// This function has been automatically generated from the project information.
{attribute 'signature_flag' := '1073741824'}
{attribute 'TcGenerated'}
{attribute 'no-analysis'}
FUNCTION F_GetTitle : WSTRING
VAR_INPUT
	
END_VAR

F_GetTitle := "ControlAlgorithm";

END_FUNCTION

(* stored: Version 1.1.0.1
   POU F_GetTitle: Id {832120c0-0328-405b-96d6-0cbefee14c2c}, SpecialFunc None *)
